(* PLC project SafeLOGIC, BrAutomation SafeDESIGNER  5.24.1.0 *)
(* stored: companyURL http://www.br-automation.com, creationDateTime Mon Dec 15 17:40:14 2025 *)

PROGRAM SCALE_AI
  VAR  (* added by the conversion: wires and edge detectors of the diagram *)
    _AND_S69_OUT : SAFEDINT;
    _ADD_S20_OUT : SAFEDINT;
  END_VAR

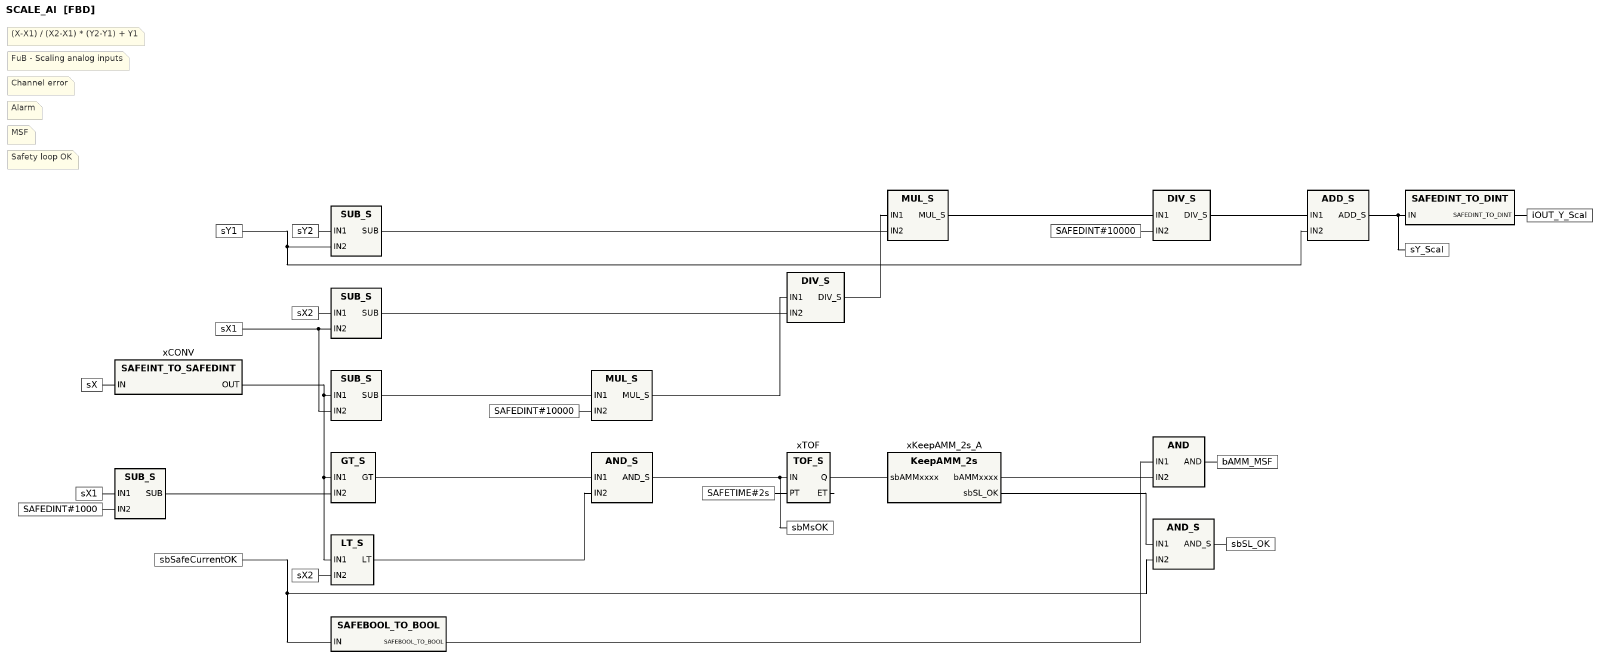
(* FBD diagram, written out as Structured Text *)
(* FuB - Scaling analog inputs *)
(* (X-X1) / (X2-X1) * (Y2-Y1) + Y1 *)
(* Alarm *)
(* Channel error *)
xCONV(IN := sX);
_AND_S69_OUT := AND_S(GT_S(xCONV.OUT, SUB_S(sX1, SAFEDINT#1000)), LT_S(xCONV.OUT, sX2));
xTOF(IN := _AND_S69_OUT, PT := SAFETIME#2s);
xKeepAMM_2s_A(sbAMMxxxx := xTOF.Q);
bAMM_MSF := SAFEBOOL_TO_BOOL(sbSafeCurrentOK) AND xKeepAMM_2s_A.bAMMxxxx;
(* Safety loop OK *)
sbSL_OK := AND_S(xKeepAMM_2s_A.sbSL_OK, sbSafeCurrentOK);
(* MSF *)
sbMsOK := _AND_S69_OUT;
_ADD_S20_OUT := ADD_S(DIV_S(MUL_S(DIV_S(MUL_S(SUB_S(xCONV.OUT, sX1), SAFEDINT#10000), SUB_S(sX2, sX1)), SUB_S(sY2, sY1)), SAFEDINT#10000), sY1);
sY_Scal := _ADD_S20_OUT;
iOUT_Y_Scal := SAFEDINT_TO_DINT(_ADD_S20_OUT);
END_PROGRAM
